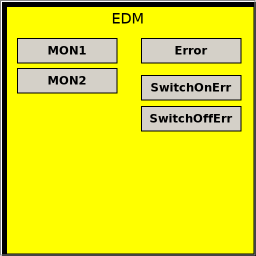
VISUALIZATION V_PH_EDM  // 256x256
VAR_INPUT
	stSafetyEDM				:ST_SAFETY_FBEDM;
	
	
END_VAR
    Rectangle (2,2 256x256), colour toggle: stSafetyEDM.bGeneralError
    Label (5,6 246x25), "EDM"
    RoundedRectangle (17,38 100x25), "MON1", colour toggle: stSafetyEDM.uStatus.stStatusWords.wInputs.8
    RoundedRectangle (141,38 100x25), "Error", colour toggle: stSafetyEDM.uStatus.stStatusWords.wOutputs.0
    RoundedRectangle (17,68 100x25), "MON2", colour toggle: stSafetyEDM.uStatus.stStatusWords.wInputs.9
    RoundedRectangle (141,106 100x25), "SwitchOffErr", colour toggle: stSafetyEDM.uStatus.stStatusWords.wDiagnosis.0, invisible if: NOT stSafetyEDM.uStatus.stStatusWords.wDiagnosis.0
    RoundedRectangle (141,75 100x25), "SwitchOnErr", colour toggle: stSafetyEDM.uStatus.stStatusWords.wDiagnosis.1, invisible if: NOT stSafetyEDM.uStatus.stStatusWords.wDiagnosis.1
    Textfield (17,226 234x25), text list: 'TL_FbState', text index: stSafetyEDM.eState
END_VISUALIZATION

(* stored: Version 1.1.0.1, ProductVersion 3.1.4024.4
   Visu V_PH_EDM: Id {5f9c0a34-d8e6-4af6-a80e-de6c40f3fb06} *)
